// TIA Portal project "level control" (V17)

(* hardware
DEVICE "S71500/ET200MP-Station_1"  S7-1500 station
   slot 0: "Profilschiene_0"  6ES7 590-1***0-0AA0
   slot 1: "PLC_1"  CPU 1511-1 PN  6ES7 511-1AK00-0AB0  V1.8
   slot 2: "AI 8xU/I/RTD/TC ST_1"  AI 8xU/I/RTD/TC ST  6ES7 531-7KF00-0AB0  V2.0
   slot 3: "AI 8xU/I/RTD/TC ST_2"  AI 8xU/I/RTD/TC ST  6ES7 531-7KF00-0AB0  V2.0
   slot 4: "AI 8xU/I/RTD/TC ST_3"  AI 8xU/I/RTD/TC ST  6ES7 531-7KF00-0AB0  V2.0
   slot 5: "AI 8xU/I/RTD/TC ST_4"  AI 8xU/I/RTD/TC ST  6ES7 531-7KF00-0AB0  V2.0
   slot 6: "DI 16x24VDC BA_1"  DI 16x24VDC BA  6ES7 521-1BH10-0AA0  V1.0
*)

// ===== PLC "PLC_1"  CPU 1511-1 PN =====

VAR_GLOBAL   // PLC tag table "Standard-Variablentabelle"
   "Start" AT %I0.0 : Bool;
   "Reset" AT %I0.1 : Bool;
   "Stop" AT %I0.2 : Bool;
   "Level meter" AT %IW30 : Int;
   "Flow meter" AT %IW32 : Int;
   "Setpoint" AT %IW34 : Int;
   "Fill valve" AT %QW30 : Int;
   "Discharge valve" AT %QW32 : Int;
   "SP" AT %QW34 : Int;
   "PV" AT %QW36 : Int;
   "Start light" AT %Q0.0 : Bool;
   "Reset light" AT %Q0.1 : Bool;
   "Stop light" AT %Q0.2 : Bool;
   "system  on" AT %M0.0 : Bool;
END_VAR

DATA_BLOCK "level control"   // DB1
{ S7_Optimized_Access := 'TRUE' }
VERSION : 0.1
   VAR
      "normalized setpoint" : Real;
      "normalized level" : Real;
   END_VAR
BEGIN
END_DATA_BLOCK

FUNCTION "MHJ-PLC-Lab-Function-S71500" : Void   // FC9000, SCL
{ S7_Optimized_Access := 'TRUE' }
VERSION : 0.1
   VAR_TEMP
      Value : Byte;
      ForCounter : Int;
   END_VAR
   VAR CONSTANT
      Value_01_DW : DWord := 16#1223_5486;
      Value_02_DW : DWord := 16#A6C9_D1F5;
   END_VAR
BEGIN

   #Value:=PEEK(area := 16#82,
        dbNumber := 0,
        byteOffset := 511);
   #Value := #Value + 1;

   POKE(area := 16#82,
        dbNumber := 0,
        byteOffset := 511,
        value := #Value);

   POKE(area := 16#82,
        dbNumber := 0,
        byteOffset := 1016,
        value := #Value_01_DW);
   POKE(area := 16#82,
        dbNumber := 0,
        byteOffset := 1020,
        value := #Value_02_DW);

   FOR #ForCounter := 0 TO 63 DO
       #Value:=PEEK(area := 16#1,
            dbNumber := 0,
            byteOffset := #ForCounter);
       POKE(area := 16#81,
            dbNumber := 0,
            byteOffset := #ForCounter,
            value := #Value);
   END_FOR;
   #Value := PEEK(area := 16#1,
                  dbNumber := 0,
                  byteOffset := 512);
   POKE(area := 16#82,
        dbNumber := 0,
        byteOffset := 512,
        value := #Value);
END_FUNCTION

ORGANIZATION_BLOCK "Main"   // OB1, LAD, ProgramCycle
TITLE = "Main Program Sweep (Cycle)"
{ S7_Optimized_Access := 'TRUE' }
VERSION : 0.1
   VAR_INPUT
      Initial_Call : Bool;   // Initial call of this OB
      Remanence : Bool;   // =True, if remanent data are available
   END_VAR
BEGIN

REGION Network 1
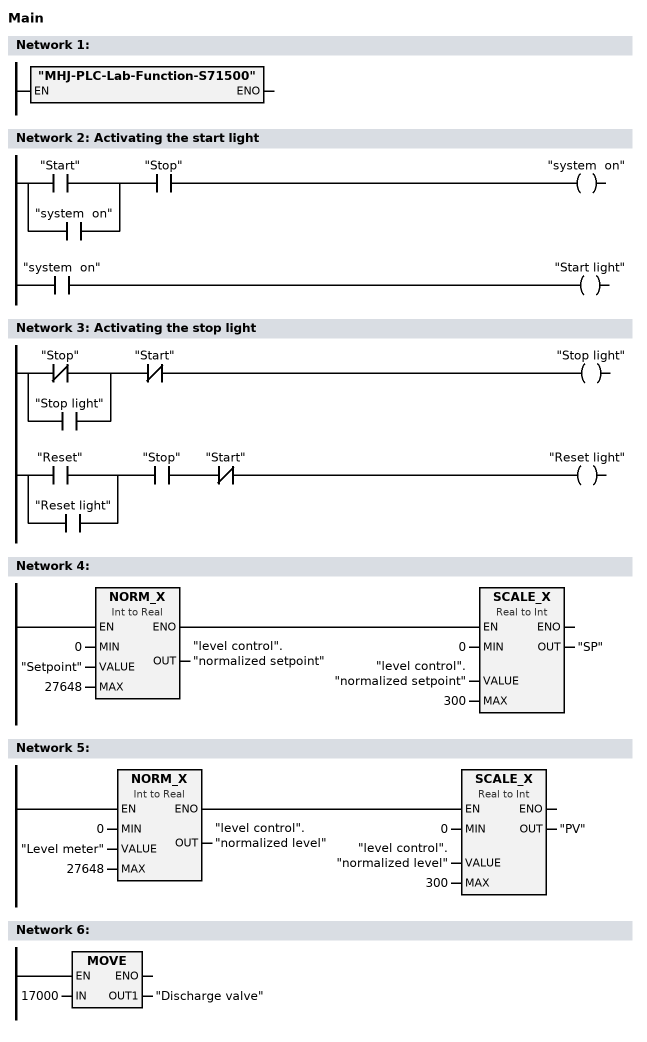
   RUNG wire#powerrail
      "MHJ-PLC-Lab-Function-S71500"()
   END_RUNG
   // the same network as SCL:
   "MHJ-PLC-Lab-Function-S71500"();
END_REGION

REGION Network 2: Activating the start light
   RUNG wire#powerrail
      Contact( "Start" )
      wire#w1
      Contact( "Stop" )
      Coil( "system  on" )
   END_RUNG
   RUNG wire#powerrail
      Contact( "system  on" )
   END_RUNG wire#w1
   RUNG wire#powerrail
      Contact( "system  on" )
      Coil( "Start light" )
   END_RUNG
   // the same network as SCL:
   "system  on" := ("Start" OR "system  on") AND "Stop";
   "Start light" := "system  on";
END_REGION

REGION Network 3: Activating the stop light
   RUNG wire#powerrail
      I_Contact( "Stop" )
      wire#w1
      I_Contact( "Start" )
      Coil( "Stop light" )
   END_RUNG
   RUNG wire#powerrail
      Contact( "Stop light" )
   END_RUNG wire#w1
   RUNG wire#powerrail
      Contact( "Reset" )
      wire#w2
      Contact( "Stop" )
      I_Contact( "Start" )
      Coil( "Reset light" )
   END_RUNG
   RUNG wire#powerrail
      Contact( "Reset light" )
   END_RUNG wire#w2
   // the same network as SCL:
   "Stop light" := (NOT "Stop" OR "Stop light") AND NOT "Start";
   "Reset light" := ("Reset" OR "Reset light") AND "Stop" AND NOT "Start";
END_REGION

REGION Network 4
   RUNG wire#powerrail
      { S7_Templates := "[SrcType := Int, DestType := Real]" } Normalize(min := 0, value := "Setpoint", max := 27648, out => "level control"."normalized setpoint")
      { S7_Templates := "[SrcType := Real, DestType := Int]" } Scale(min := 0, value := "level control"."normalized setpoint", max := 300, out => "SP")
   END_RUNG
   // the same network as SCL:
   "level control"."normalized setpoint" := NORM_X(MIN := 0, VALUE := "Setpoint", MAX := 27648);
   "SP" := SCALE_X(MIN := 0, VALUE := "level control"."normalized setpoint", MAX := 300);
END_REGION

REGION Network 5
   RUNG wire#powerrail
      { S7_Templates := "[SrcType := Int, DestType := Real]" } Normalize(min := 0, value := "Level meter", max := 27648, out => "level control"."normalized level")
      { S7_Templates := "[SrcType := Real, DestType := Int]" } Scale(min := 0, value := "level control"."normalized level", max := 300, out => "PV")
   END_RUNG
   // the same network as SCL:
   "level control"."normalized level" := NORM_X(MIN := 0, VALUE := "Level meter", MAX := 27648);
   "PV" := SCALE_X(MIN := 0, VALUE := "level control"."normalized level", MAX := 300);
END_REGION

REGION Network 6
   RUNG wire#powerrail
      Move(in := 17000, out1 => "Discharge valve")
   END_RUNG
   // the same network as SCL:
   "Discharge valve" := 17000;
END_REGION
END_ORGANIZATION_BLOCK

ORGANIZATION_BLOCK "Cyclic interrupt"   // OB30, LAD, CyclicInterrupt
{ S7_Optimized_Access := 'TRUE' }
VERSION : 0.1
   VAR_INPUT
      Initial_Call : Bool;   // Initial call of this OB
      Event_Count : Int;   // Events discarded
   END_VAR
BEGIN

REGION Network 1
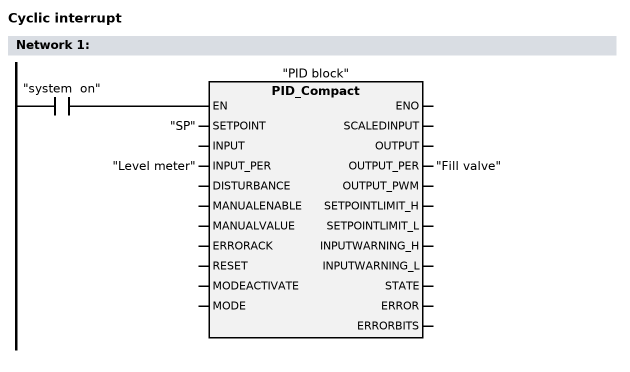
   IF "system  on" THEN
       "PID block"(Setpoint := "SP", Input_PER := "Level meter", Output_PER => "Fill valve");   // PID_Compact
   END_IF;
END_REGION
END_ORGANIZATION_BLOCK